// TIA Portal V19 export
DATA_BLOCK "Bottom_Valve_Control"   // DB2
// stored: InstanceOfName Vavle_Control, InstanceOfType FB
"Vavle_Control"
   // VAR_INPUT
   //    Closed : Bool;
   //    Open : Bool;
   //    OpenValve : Bool;
   // END_VAR
   // VAR_OUTPUT
   //    Actuator : Bool;
   //    State : String;
   //    StateNum : Int;
   // END_VAR
   // VAR
   //    OldOpenValve : Bool;
   // END_VAR
BEGIN
END_DATA_BLOCK
